{attribute addProperty BoxType "ELM3002-0000-0016"}
{attribute addProperty Id "No_of_SamplesUSINT811ErrorBIT10.1259UnderrangeBIT10.12510OverrangeBIT10.12511DiagBIT10.12513TxPDO_StateBIT10.12514Input_cycle_counter_BIT_0BIT10.12515Input_cycle_counter_BIT_1BIT10.12515"}
{attribute addProperty CRC "1782636244"}
{attribute addProperty SizeInBites "32"}
{attribute addProperty SizeInBytes "4"}
TYPE Status_6A40DED4 :
STRUCT
	{attribute addProperty Name "No_of_Samples"}
	No_of_Samples : USINT;
	{attribute addProperty Name "Error"}
	Error : BIT;
	{attribute addProperty Name "Underrange"}
	Underrange : BIT;
	{attribute addProperty Name "Overrange"}
	Overrange : BIT;
	{attribute 'hide'}
	reserve_1 : BIT;
	{attribute addProperty Name "Diag"}
	Diag : BIT;
	{attribute addProperty Name "TxPDO_State"}
	TxPDO_State : BIT;
	{attribute addProperty Name "Input_cycle_counter"}
	Input_cycle_counter_BIT_0 : BIT;
	{attribute addProperty Name "Input_cycle_counter"}
	Input_cycle_counter_BIT_1 : BIT;
	{attribute 'hide'}
	reserve_2_BYTE_0 : BYTE;
	{attribute 'hide'}
	reserve_2_BYTE_1 : BYTE;
END_STRUCT
END_TYPE

(* stored: Version 1.2.0.0, ProductVersion 3.1.4024.9
   DUT Status_6A40DED4: Id {13ab1308-63fb-4ba5-a1ea-0c68d5c5cebb} *)
